PROGRAM MAIN
VAR
	MyBoolean : BOOL;
	
	bRunMath : BOOL;
	
	iValue1 : DINT := 20;
	iValue2 : DINT;
	
	i : INT;
	j : INT;
	c : DINT;
	
	sMyString : STRING;
	sMyNumString : STRING[255];
	
	i_Num_from_arr : DINT;
	i_len_arr_B : INT;
	arr_A : ARRAY [0..10] OF DINT;
	arr_B : ARRAY [0..4] OF DINT :=[20, 40, 60 ,80, 100];
	
	// timers
	fb_My_timer : TON;
	// tiggers
	fb_my_trigger : R_TRIG; // Counter 
	
	// Timer
	fb_MI1_Timer_Increase_Speed: TON;
	
	// Speed setup
	f_MI1_Initial_Speed: REAL := 20;
	f_MI1_Constant_Speed: REAL := 60;
	f_MI1_Max_Speed : REAL := 120;
END_VAR

VAR_OUTPUT
	// Speed Output
	f_MI1_Speed: REAL;
END_VAR


f_MI1_Speed:= f_MI1_Initial_Speed;

IF MyBoolean THEN
	REPEAT
		fb_MI1_Timer_Increase_Speed(
			IN:=MyBoolean,
			PT:= T#20S);
		IF fb_MI1_Timer_Increase_Speed.Q THEN
			f_MI1_Speed := f_MI1_Speed + f_MI1_Initial_Speed;
		END_IF
		
	UNTIL 
		f_MI1_Speed > 120 
	END_REPEAT
	
END_IF

END_PROGRAM

(* stored: Version 1.1.0.1, ProductVersion 3.1.4024.11
   POU MAIN: Id {38e7ac3d-a4b5-4c4e-904d-27c6290e435e}, SpecialFunc None *)
